(* LS Electric XG5000 project: 제일교회_조명제어 *)
(* PLC LSPLC *)
(* module base 0 slot 0: Cnet:XGL-C42A/B (Cnet 통신 모듈(RS-422/485, RS-422/485)) *)
(* module base 0 slot 1: 입력 모듈:XGI-D24A/B (DC 24V 입력, 32점 (전류소스 싱크공용/ 전류소스 입력)) *)
(* module base 0 slot 2: 입력 모듈:XGI-D21A (DC 24V 입력, 8점 (전류소스/싱크입력)) *)
(* module base 0 slot 3: 출력 모듈:XGQ-TR4A/B (트랜지스터 출력, 32점 (0.1A용, 싱크출력/소스출력)) *)

(* Comments on direct variables
%MX92	SET - 01_Button
%MX93	SET - 02_Button
%MX94	SET - 03_Button
%MX95	SET - 01_Lamp
%MX96	SET - 02_Lamp
%MX97	SET - 03_Lamp
%MX98	Reset
[SCADA]
%MX99	SHUT OFF
%MX100	MAIN POWER PBL
%MX101	십자가 PBL
%MX102	강대상 위 천정 PBL
%MX103	강대석(좌) PBL
%MX104	무대조명(좌) PBL
%MX105	(미정) PBL
%MX106	본당벽체 간접 PBL
%MX107	복도(좌) PBL
%MX108	중벽체(반달 좌) PBL
%MX109	중벽체 간접(좌) PBL
%MX110	기둥간접(좌) PBL
%MX111	중앙천정 강대상 PBL
%MX112	중앙천정앞(50W전구색) PBL
%MX113	중앙천정좌 간접 PBL
%MX114	중앙천정우 간접 PBL
%MX115	중앙천정U(20W주광색) PBL
%MX116	중앙천정뒤(50W전구색) PBL
%MX117	강대석 (우) PBL
%MX118	무대조명(우) PBL
%MX119	(미정) PBL
%MX120	본당벽체 간접 PBL
%MX121	복도(우) PBL
%MX122	중벽채(반달 우) PBL
%MX123	중벽체 간접(우) PBL
%MX124	기둥간접(우) PBL
%MX125	2층 후미 PBL
%MX126	종탑 PBL
%MX127	LAMP TEST PBL
%MX128	BUZZER STOP PBL[SR]
%MX129	RESET PBL[SR]
%MX130	SPARE
%MX131	SPARE
%MX160	Main Switch On
%MX161	성가대 P-S/W
%MX170	SCADA POWER PB [SCA]
%MX171	REMOTE POWER PB [SCA]
%MX192	십자가_SET [SCADA]
%MX193	강대상 위 천장_SET [SCADA]
%MX194	강대석 좌_SET [SCADA]
%MX195	무대조명(좌)_SET [SCADA]
%MX197	본당벽체-간접(좌)_SET [SCADA]
%MX198	복도(좌)_SET [SCADA]
%MX199	중벽체-반달(좌)_SET [SCADA]
%MX200	중벽체-간접(좌)_SET [SCADA]
%MX202	중앙천장 강대상_SET [SCADA]
%MX203	중앙천장앞_SET [SCADA]
%MX204	중앙천정좌 간접_SET [SCADA]
%MX205	중앙천장우 간접_SET [SCADA]
%MX206	중앙천정 U_SET [SCADA]
%MX207	중앙천정-뒤_SET [SCADA]
%MX208	강대석-우_SET [SCADA]
%MX209	무대조명(우)_SET [SCADA]
%MX211	본당벽체-간접(우)_SET [SCADA]
%MX212	복도(우)_SET [SCADA]
%MX213	중벽체-반달(우)_SET [SCADA]
%MX214	중벽체-간접 (우)_SET [SCADA]
%MX216	후미 중앙 기둥 간접등_SET [SCADA]
%MX217	종탑_SET [SCADA]
%MX284	BUZZER STOP [SCA]
%MX400	REMOTE POWER LAMP[REM]
%MX401	십자가 [REM]
%MX402	강대상 위 천정 [REM]
%MX403	강대석(좌) [REM]
%MX404	무대조명(좌) [REM]
%MX405	(미정) [REM]
%MX406	본당벽체 간접 [REM]
%MX407	복도 [REM]
%MX408	중벽체-반달(좌) [REM]
%MX409	중벽체 간접 [REM]
%MX410	기둥간접 [REM]
%MX411	중앙천정 강대상
[REM]
%MX412	중앙천정앞
50W전구색
[REM]
%MX413	중앙천정좌 간접 [REM]
%MX414	중앙천정우 간접 [REM]
%MX415	중앙천정U(20W주광색) [REM]
%MX416	중앙천정뒤(50W전구색) [REM]
%MX417	강대석 (우) [REM]
%MX418	무대조명(우) [REM]
%MX419	(미정) [REM]
%MX420	본당벽체 간접 [REM]
%MX421	복도 [REM]
%MX422	중벽채-반달(우) [REM]
%MX423	중벽체 간접 [REM]
%MX424	기둥간접 [REM]
%MX425	2층 후미 [REM]
%MX426	종탑 [REM]
%MX427	LAMP TEST [REM]
%MX428	BUZZER STOP [REM]
%MX429	RESET [REM]
%MX430	SPARE [REM]
%MX431	SPARE [REM]
%MX500	MAIN POWER LAMP
%MX501	십자가 LAMP
%MX502	강대상 위 천정 LAMP
%MX503	강대석(좌) LAMP
%MX504	무대조명(좌) LAMP
%MX505	(미정) LAMP
%MX506	본당벽체 간접 LAMP
%MX507	복도 LAMP
%MX508	중벽체(반달) LAMP
%MX509	중벽체 간접 LAMP
%MX510	기둥간접 LAMP
%MX511	중앙천정 강대상 LAMP
%MX512	중앙천정앞(50W전구색) LAMP
%MX513	중앙천정좌 간접 LAMP
%MX514	중앙천정우 간접 LAMP
%MX515	중앙천정U(20W주광색) LAMP
%MX516	중앙천정뒤(50W전구색) LAMP
%MX517	강대석 (우) LAMP
%MX518	무대조명(우) LAMP
%MX519	(미정) LAMP
%MX520	본당벽체 간접 LAMP
%MX521	복도 LAMP
%MX522	중벽채(반달) LAMP
%MX523	중벽체 간접 LAMP
%MX524	기둥간접 LAMP
%MX525	2층 후미 LAMP
%MX526	종탑 LAMP
%MX527	LAMP TEST LAMP
%MX528	BUZZER STOP LAMP
%MX529	RESET LAMP
%MX530	BUZZER
[[REM]]
%MX531	SPARE LAMP
%MX600	SCADA POWER LAMP_[SCA]
%MX601	십자가_S/W [SCADA]
%MX602	강대상 위 천장_S/W [SCADA]
%MX603	강대석 좌_S/W [SCADA]
%MX604	무대조명(좌)_S/W [SCADA]
%MX606	본당벽체-간접(좌)_S/W [SCADA]
%MX607	복도(좌)_S/W [SCADA]
%MX608	중벽체-반달(좌)_S/W [SCADA]
%MX609	중벽체-간접(좌)_S/W [SCADA]
%MX611	중앙천장 강대상_S/W [SCADA]
%MX612	중앙천장앞_S/W [SCADA]
%MX613	중앙천정좌 간접_S/W [SCADA]
%MX614	중앙천장우 간접_S/W [SCADA]
%MX615	중앙천정 U_S/W [SCADA]
%MX616	중앙천정-뒤_S/W [SCADA]
%MX617	강대석-우_S/W [SCADA]
%MX618	무대조명(우)_S/W [SCADA]
%MX620	본당벽체-간접(우)_S/W [SCADA]
%MX621	복도(우)_S/W [SCADA]
%MX622	중벽체-반달(우)_S/W [SCADA]
%MX623	중벽체-간접 (우)_S/W [SCADA]
%MX625	후미 중앙 기둥 간접등_S/W [SCADA]
%MX626	종탑_S/W [SCADA]
%MX640	중앙1열 OUT
%MX641	중앙2열 OUT
%MX642	중앙3열 OUT
%MX643	중앙4열 OUT
%MX644	중앙5열 OUT
%MX645	중앙6열 OUT
%MX646	중앙7열 OUT
%MX647	중앙8열 OUT
%MX648	중앙9열 OUT
%MX649	중앙10열 OUT
%MX650	장로석 OUT
%MX651	장로석 SPOT-OUT
%MX652	성가대 OUT
%MX653	성가대 SPOT-OUT
%MX654	좌측통로 OUT
%MX655	우측통로 OUT
%MX656	후단1열 OUT
%MX657	후단2열 OUT
%MX658	후단3열 OUT
%MX659	종탑 OUT
%MX704	십자가_[SET]_OUT [SCADA]
%MX705	강대상 위 천장_[SET]_OUT [SCADA]
%MX706	강대석 좌_[SET]_OUT [SCADA]
%MX707	무대조명(좌)_[SET]_OUT [SCADA]
%MX709	본당벽체-간접(좌)_[SET]_OUT [SCADA]
%MX710	복도(좌)_[SET]_OUT [SCADA]
%MX711	중벽체-반달(좌)_[SET]_OUT [SCADA]
%MX712	중벽체-간접(좌)_[SET]_OUT [SCADA]
%MX714	중앙천장 강대상_[SET]_OUT [SCADA]
%MX715	중앙천장앞_[SET]_OUT [SCADA]
%MX716	중앙천정좌 간접_[SET]_OUT [SCADA]
%MX717	중앙천장우 간접_[SET]_OUT [SCADA]
%MX718	중앙천정 U_[SET]_OUT [SCADA]
%MX719	중앙천정-뒤_[SET]_OUT [SCADA]
%MX720	강대석-우_[SET]_OUT [SCADA]
%MX721	무대조명(우)_[SET]_OUT [SCADA]
%MX723	본당벽체-간접(우)_[SET]_OUT [SCADA]
%MX724	복도(우)_[SET]_OUT [SCADA]
%MX725	중벽체-반달(우)_[SET]_OUT [SCADA]
%MX726	중벽체-간접 (우)_[SET]_OUT [SCADA]
%MX728	후미 중앙 기둥 간접등_[SET]_OUT [SCADA]
%MX729	종탑_[SET]_OUT [SCADA]
%MX800	십자가_S/W_OUT [SCADA]
%MX801	강대상 위 천장_S/W_OUT [SCADA]
%MX802	강대석 좌_S/W_OUT [SCADA]
%MX803	무대조명(좌)_S/W_OUT [SCADA]
%MX805	본당벽체-간접(좌)_S/W_OUT [SCADA]
%MX806	복도(좌)_S/W_OUT [SCADA]
%MX807	중벽체-반달(좌)_S/W_OUT [SCADA]
%MX808	중벽체-간접(좌)_S/W_OUT [SCADA]
%MX810	중앙천장 강대상_S/W_OUT [SCADA]
%MX811	중앙천장앞_S/W_OUT [SCADA]
%MX812	중앙천정좌 간접_S/W_OUT [SCADA]
%MX813	중앙천장우 간접_S/W_OUT [SCADA]
%MX814	중앙천정 U_S/W_OUT [SCADA]
%MX815	중앙천정-뒤_S/W_OUT [SCADA]
%MX816	강대석-우_S/W_OUT [SCADA]
%MX817	무대조명(우)_S/W_OUT [SCADA]
%MX819	본당벽체-간접(우)_S/W_OUT [SCADA]
%MX820	복도(우)_S/W_OUT [SCADA]
%MX821	중벽체-반달(우)_S/W_OUT [SCADA]
%MX822	중벽체-간접 (우)_S/W_OUT [SCADA]
%MX824	후미 중앙 기둥 간접등_S/W_OUT [SCADA]
%MX825	종탑_S/W_OUT [SCADA]
%MX911	Total Alarm
%MX992	중앙1열 S/W
%MX993	중앙2열 S/W
%MX994	중앙3열 S/W
%MX995	중앙4열 S/W
%MX996	중앙5열 S/W
%MX997	중앙6열 S/W
%MX998	중앙7열 S/W
%MX999	중앙8열 S/W
%MX1000	중앙9열 S/W
%MX1001	중앙10열 S/W
%MX1002	장로석 S/W
%MX1003	장로석 SPOT S/W
%MX1004	성가대 S/W
%MX1005	성가대 SPOT S/W [MAIN]
%MX1006	좌측통로 S/W
%MX1007	우측통로 S/W
%MX1008	후단1열 S/W
%MX1009	후단2열 S/W
%MX1010	후단3열 S/W
%MX1011	종탑 S/W
%MX1040	중앙1열 M/C-a
%MX1041	중앙2열 M/C-a
%MX1042	중앙3열 M/C-a
%MX1043	중앙4열 M/C-a
%MX1044	중앙5열 M/C-a
%MX1045	중앙6열 M/C-a
%MX1046	중앙7열 M/C-a
%MX1047	중앙8열 M/C-a
%MX1048	중앙9열 M/C-a
%MX1049	중앙10열 M/C-a
%MX1050	장로석 M/C-a
%MX1051	장로석 SPOT M/C-a
%MX1052	성가대 M/C-a
%MX1053	성가대 SPOT M/C-a
%MX1054	좌측통로 M/C-a
%MX1055	우측통로 M/C-a
%MX1056	후단1열 M/C-a
%MX1057	후단2열 M/C-a
%MX1058	후단3열 M/C-a
%MX1059	종탑 M/C-a
%MW0	IN-COM0
%MW1	IN-COM1
%MW2	OUT-COM0
%MW3	OUT-COM1
%MW4	Reset-Word
%MW12	Reset-Word
%MD22	SET_OUT
%MD31	MAIN_SW
%QX0.3.0	중앙1열
%QX0.3.1	중앙2열
%QX0.3.2	중앙3열
%QX0.3.3	중앙4열
%QX0.3.4	중앙5열
%QX0.3.5	중앙6열
%QX0.3.6	중앙7열
%QX0.3.7	중앙8열
%QX0.3.8	중앙9열
%QX0.3.9	중앙10열
%QX0.3.10	장로석
%QX0.3.11	장로석 SPOT
%QX0.3.12	성가대
%QX0.3.13	성가대 SPOT
%QX0.3.14	좌측통로
%QX0.3.15	우측통로
%QX0.3.16	후단1열
%QX0.3.17	후단2열
%QX0.3.18	후단3열
%QX0.3.19	종탑
%QX0.3.20	BUZZER
[MAIN]
%IX0.1.0	중앙1열 S/W
%IX0.1.1	중앙2열 S/W
%IX0.1.2	중앙3열 S/W
%IX0.1.3	중앙4열 S/W
%IX0.1.4	중앙5열 S/W
%IX0.1.5	중앙6열 S/W
%IX0.1.6	중앙7열 S/W
%IX0.1.7	중앙8열 S/W
%IX0.1.8	중앙9열 S/W
%IX0.1.9	중앙10열 S/W
%IX0.1.10	장로석 S/W
%IX0.1.11	장로석 SPOT S/W
%IX0.1.12	성가대 S/W
%IX0.1.13	성가대 SPOT S/W
%IX0.1.14	좌측통로 S/W
%IX0.1.15	우측통로 S/W
%IX0.1.16	후단1열 S/W
%IX0.1.17	후단2열 S/W
%IX0.1.18	후단3열 S/W
%IX0.1.19	종탑
%IX0.1.20	중앙1열 M/C-a
%IX0.1.21	중앙2열 M/C-a
%IX0.1.22	중앙3열 M/C-a
%IX0.1.23	중앙4열 M/C-a
%IX0.1.24	중앙5열 M/C-a
%IX0.1.25	중앙6열 M/C-a
%IX0.1.26	중앙7열 M/C-a
%IX0.1.27	중앙8열 M/C-a
%IX0.1.28	중앙9열 M/C-a
%IX0.1.29	중앙10열 M/C-a
%IX0.1.30	장로석 M/C-a
%IX0.1.31	장로석 SPOT M/C-a
%IX0.2.0	성가대 M/C-a
%IX0.2.1	성가대 SPOT M/C-a
%IX0.2.2	좌측통로 M/C-a
%IX0.2.3	우측통로 M/C-a
%IX0.2.4	후단1열 M/C-a
%IX0.2.5	후단2열 M/C-a
%IX0.2.6	후단3열 M/C-a
%IX0.2.7	종탑
M/C-a
*)

FUNCTION_BLOCK SET_FF
VAR_INPUT
    IN : BOOL;
    RESET : BOOL;
    CHECK_SET : BOOL;
END_VAR
VAR_IN_OUT
    SET : BOOL;
    MANUAL : BOOL;
END_VAR
VAR_OUTPUT
    FF : BOOL;
END_VAR
VAR
    IN_COIL : BOOL;
END_VAR
VAR
    _e1 : R_TRIG;
    _e2 : R_TRIG;
END_VAR

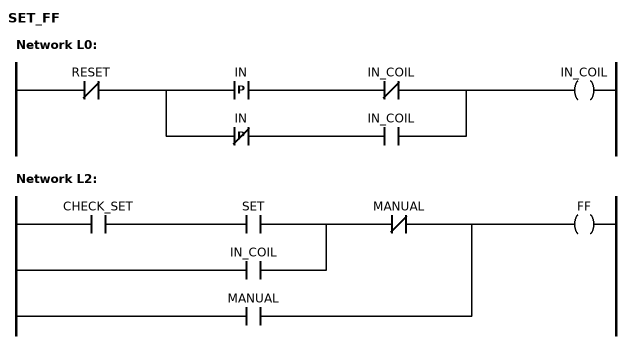
(* Rung L0 *)
_e1(CLK := IN);
_e2(CLK := IN);
IN_COIL := NOT RESET AND ((_e1.Q AND NOT IN_COIL) OR (NOT _e2.Q AND IN_COIL));
(* Rung L2 *)
FF := (((CHECK_SET AND SET) OR IN_COIL) AND NOT MANUAL) OR MANUAL;
END_FUNCTION_BLOCK

PROGRAM Remote (* task: 스캔 프로그램 *)
VAR
    INST : FF;
    INST1 : FF;
    IN_0_HIGH : BYTE;
    IN_0_LOW : BYTE;
    IN_1_HIGH : BYTE;
    IN_1_LOW : BYTE;
    OUT_0_HIGH : BYTE;
    OUT_0_LOW : BYTE;
    remote_holding : BOOL;
END_VAR

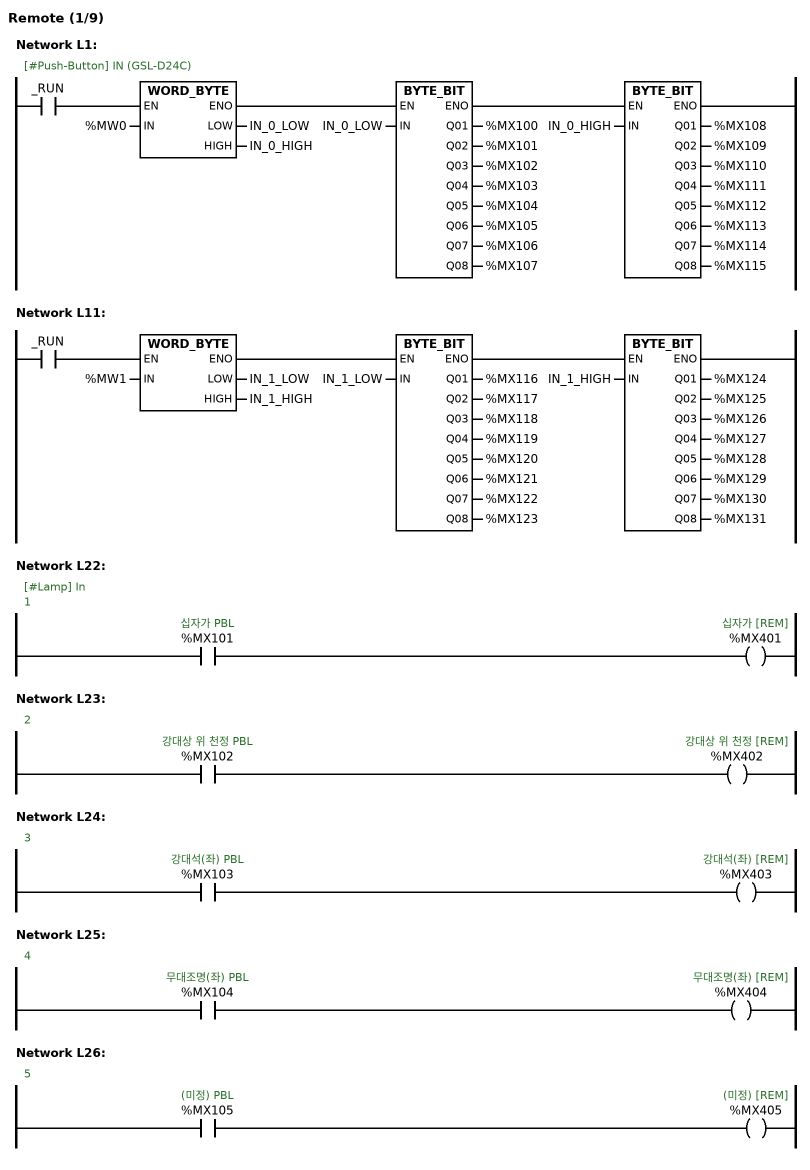
(* [#Push-Button] IN (GSL-D24C) *)
(* Rung L1 *)
IF _RUN THEN
    IN_0_LOW := WORD_BYTE(IN := %MW0, HIGH => IN_0_HIGH);
    %MX100 := BYTE_BIT(IN := IN_0_LOW, Q02 => %MX101, Q03 => %MX102, Q04 => %MX103, Q05 => %MX104, Q06 => %MX105, Q07 => %MX106, Q08 => %MX107);
    %MX108 := BYTE_BIT(IN := IN_0_HIGH, Q02 => %MX109, Q03 => %MX110, Q04 => %MX111, Q05 => %MX112, Q06 => %MX113, Q07 => %MX114, Q08 => %MX115);
END_IF;
(* Rung L11 *)
IF _RUN THEN
    IN_1_LOW := WORD_BYTE(IN := %MW1, HIGH => IN_1_HIGH);
    %MX116 := BYTE_BIT(IN := IN_1_LOW, Q02 => %MX117, Q03 => %MX118, Q04 => %MX119, Q05 => %MX120, Q06 => %MX121, Q07 => %MX122, Q08 => %MX123);
    %MX124 := BYTE_BIT(IN := IN_1_HIGH, Q02 => %MX125, Q03 => %MX126, Q04 => %MX127, Q05 => %MX128, Q06 => %MX129, Q07 => %MX130, Q08 => %MX131);
END_IF;
(* [#Lamp] In *)
(* Rung L22 *)
%MX401 := %MX101;
(* 1 *)
(* Rung L23 *)
%MX402 := %MX102;
(* 2 *)
(* Rung L24 *)
%MX403 := %MX103;
(* 3 *)
(* Rung L25 *)
%MX404 := %MX104;
(* 4 *)
(* Rung L26 *)
%MX405 := %MX105;
(* 5 *)

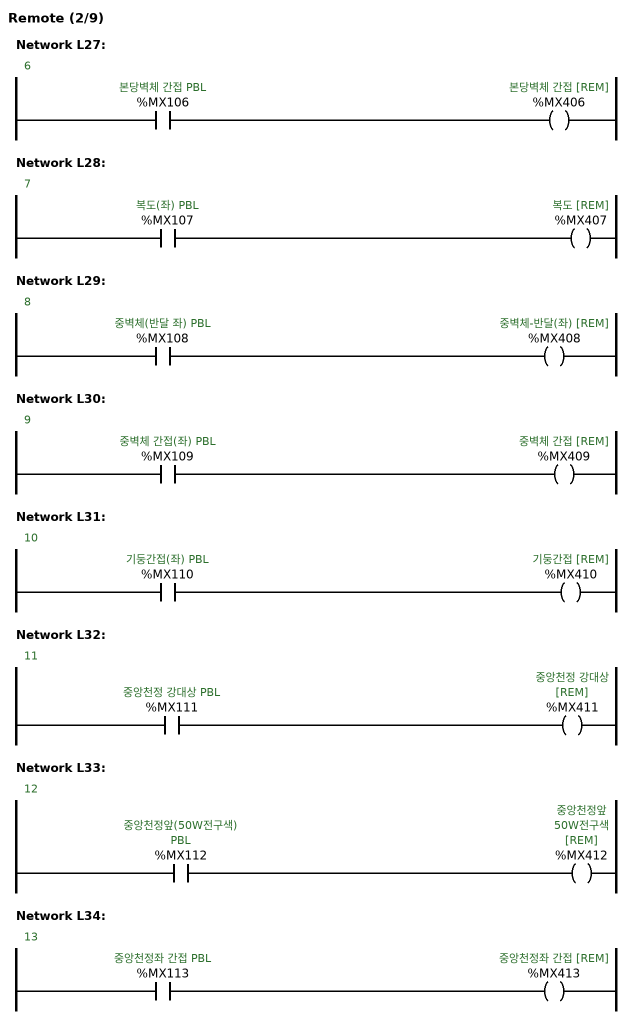
(* Rung L27 *)
%MX406 := %MX106;
(* 6 *)
(* Rung L28 *)
%MX407 := %MX107;
(* 7 *)
(* Rung L29 *)
%MX408 := %MX108;
(* 8 *)
(* Rung L30 *)
%MX409 := %MX109;
(* 9 *)
(* Rung L31 *)
%MX410 := %MX110;
(* 10 *)
(* Rung L32 *)
%MX411 := %MX111;
(* 11 *)
(* Rung L33 *)
%MX412 := %MX112;
(* 12 *)
(* Rung L34 *)
%MX413 := %MX113;
(* 13 *)

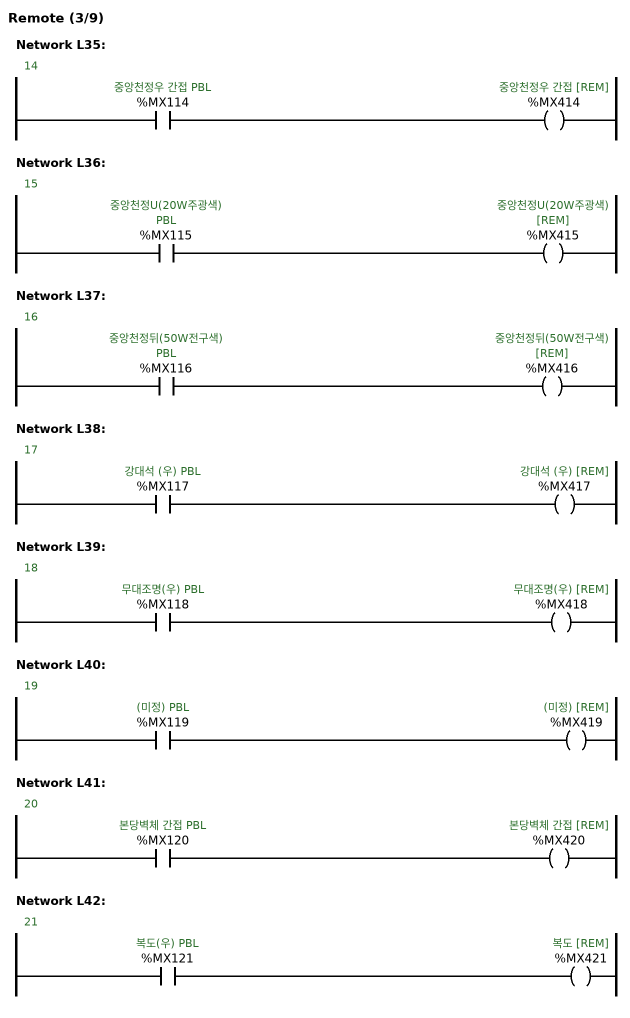
(* Rung L35 *)
%MX414 := %MX114;
(* 14 *)
(* Rung L36 *)
%MX415 := %MX115;
(* 15 *)
(* Rung L37 *)
%MX416 := %MX116;
(* 16 *)
(* Rung L38 *)
%MX417 := %MX117;
(* 17 *)
(* Rung L39 *)
%MX418 := %MX118;
(* 18 *)
(* Rung L40 *)
%MX419 := %MX119;
(* 19 *)
(* Rung L41 *)
%MX420 := %MX120;
(* 20 *)
(* Rung L42 *)
%MX421 := %MX121;
(* 21 *)

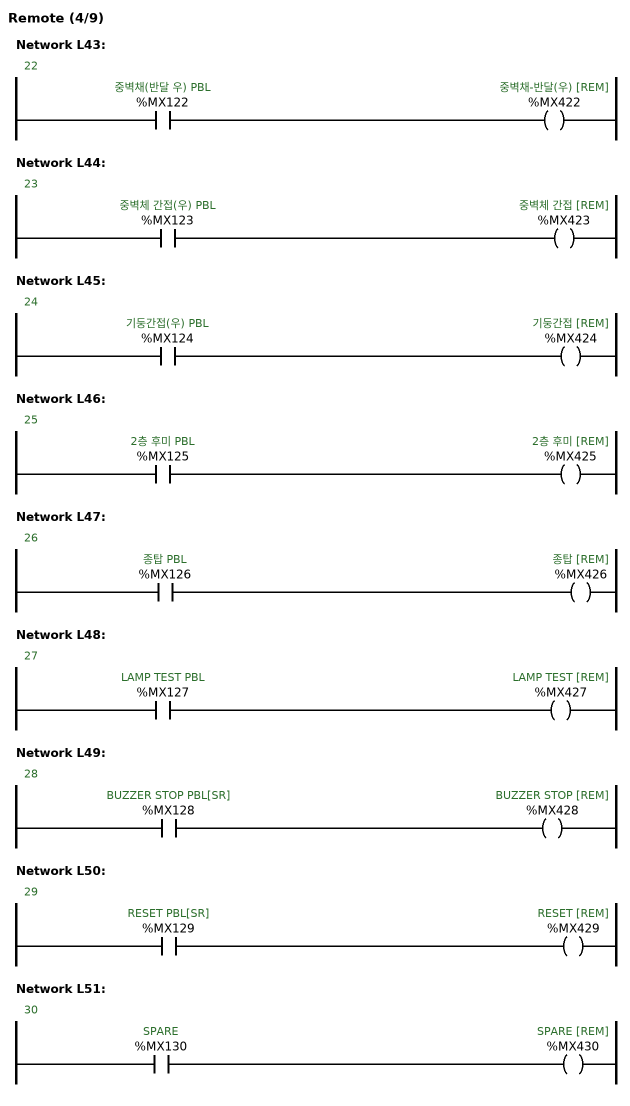
(* Rung L43 *)
%MX422 := %MX122;
(* 22 *)
(* Rung L44 *)
%MX423 := %MX123;
(* 23 *)
(* Rung L45 *)
%MX424 := %MX124;
(* 24 *)
(* Rung L46 *)
%MX425 := %MX125;
(* 25 *)
(* Rung L47 *)
%MX426 := %MX126;
(* 26 *)
(* Rung L48 *)
%MX427 := %MX127;
(* 27 *)
(* Rung L49 *)
%MX428 := %MX128;
(* 28 *)
(* Rung L50 *)
%MX429 := %MX129;
(* 29 *)
(* Rung L51 *)
%MX430 := %MX130;
(* 30 *)

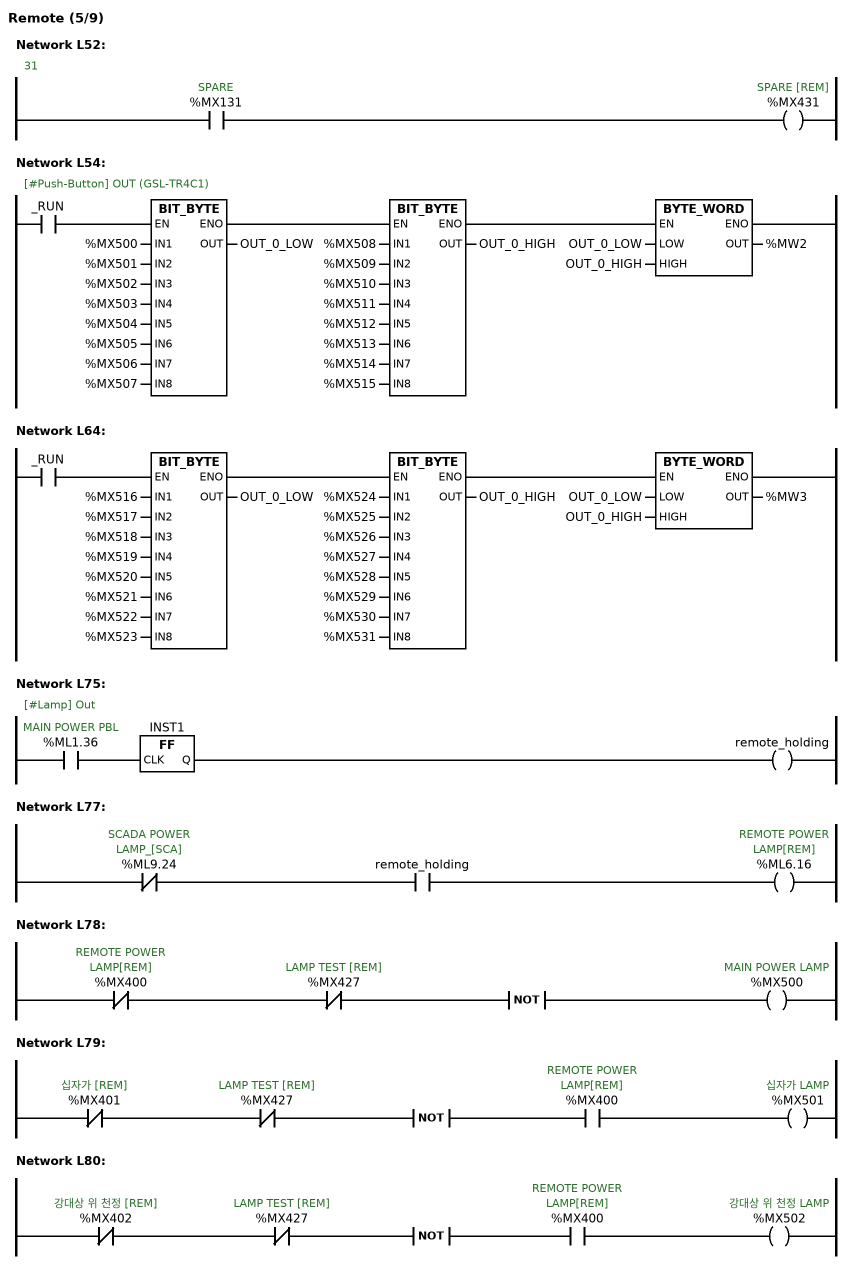
(* Rung L52 *)
%MX431 := %MX131;
(* 31 *)
(* [#Push-Button] OUT (GSL-TR4C1) *)
(* Rung L54 *)
IF _RUN THEN
    OUT_0_LOW := BIT_BYTE(%MX500, %MX501, %MX502, %MX503, %MX504, %MX505, %MX506, %MX507);
    OUT_0_HIGH := BIT_BYTE(%MX508, %MX509, %MX510, %MX511, %MX512, %MX513, %MX514, %MX515);
    %MW2 := BYTE_WORD(LOW := OUT_0_LOW, HIGH := OUT_0_HIGH);
END_IF;
(* Rung L64 *)
IF _RUN THEN
    OUT_0_LOW := BIT_BYTE(%MX516, %MX517, %MX518, %MX519, %MX520, %MX521, %MX522, %MX523);
    OUT_0_HIGH := BIT_BYTE(%MX524, %MX525, %MX526, %MX527, %MX528, %MX529, %MX530, %MX531);
    %MW3 := BYTE_WORD(LOW := OUT_0_LOW, HIGH := OUT_0_HIGH);
END_IF;
(* [#Lamp] Out *)
(* Rung L75 *)
INST1(CLK := %ML1.36);
remote_holding := INST1.Q;
(* Rung L77 *)
%ML6.16 := NOT %ML9.24 AND remote_holding;
(* Rung L78 *)
%MX500 := NOT (NOT %MX400 AND NOT %MX427);
(* Rung L79 *)
%MX501 := NOT (NOT %MX401 AND NOT %MX427) AND %MX400;
(* Rung L80 *)
%MX502 := NOT (NOT %MX402 AND NOT %MX427) AND %MX400;

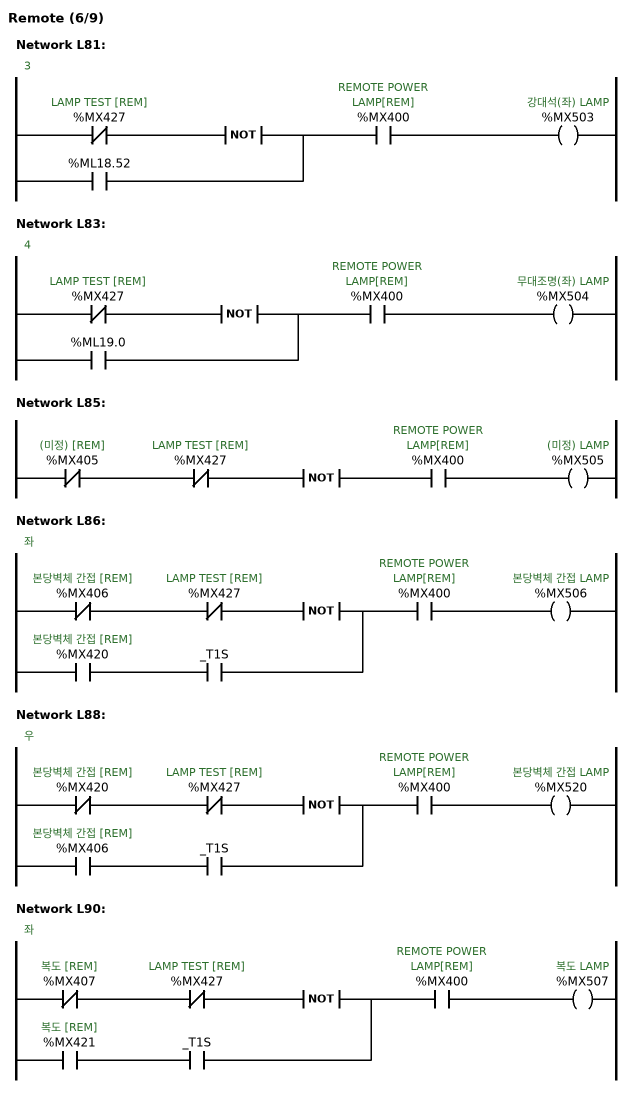
(* Rung L81 *)
%MX503 := (%MX427 OR %ML18.52) AND %MX400;
(* 3 *)
(* Rung L83 *)
%MX504 := (%MX427 OR %ML19.0) AND %MX400;
(* 4 *)
(* Rung L85 *)
%MX505 := NOT (NOT %MX405 AND NOT %MX427) AND %MX400;
(* Rung L86 *)
%MX506 := (NOT (NOT %MX406 AND NOT %MX427) OR (%MX420 AND _T1S)) AND %MX400;
(* 좌 *)
(* Rung L88 *)
%MX520 := (NOT (NOT %MX420 AND NOT %MX427) OR (%MX406 AND _T1S)) AND %MX400;
(* 우 *)
(* Rung L90 *)
%MX507 := (NOT (NOT %MX407 AND NOT %MX427) OR (%MX421 AND _T1S)) AND %MX400;
(* 좌 *)

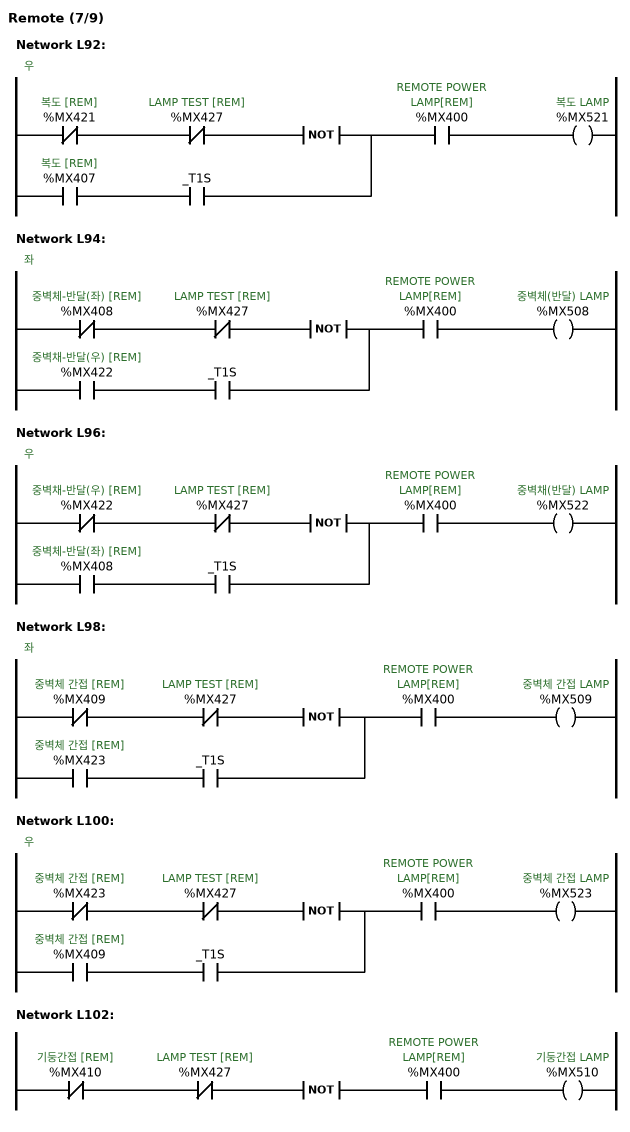
(* Rung L92 *)
%MX521 := (NOT (NOT %MX421 AND NOT %MX427) OR (%MX407 AND _T1S)) AND %MX400;
(* 우 *)
(* Rung L94 *)
%MX508 := (NOT (NOT %MX408 AND NOT %MX427) OR (%MX422 AND _T1S)) AND %MX400;
(* 좌 *)
(* Rung L96 *)
%MX522 := (NOT (NOT %MX422 AND NOT %MX427) OR (%MX408 AND _T1S)) AND %MX400;
(* 우 *)
(* Rung L98 *)
%MX509 := (NOT (NOT %MX409 AND NOT %MX427) OR (%MX423 AND _T1S)) AND %MX400;
(* 좌 *)
(* Rung L100 *)
%MX523 := (NOT (NOT %MX423 AND NOT %MX427) OR (%MX409 AND _T1S)) AND %MX400;
(* 우 *)
(* Rung L102 *)
%MX510 := NOT (NOT %MX410 AND NOT %MX427) AND %MX400;

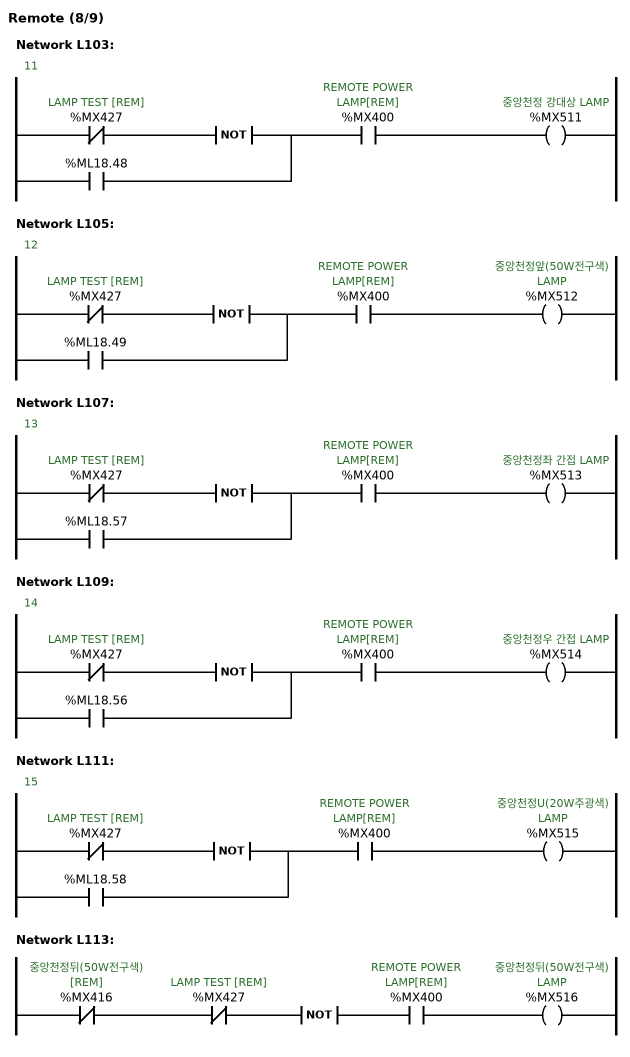
(* Rung L103 *)
%MX511 := (%MX427 OR %ML18.48) AND %MX400;
(* 11 *)
(* Rung L105 *)
%MX512 := (%MX427 OR %ML18.49) AND %MX400;
(* 12 *)
(* Rung L107 *)
%MX513 := (%MX427 OR %ML18.57) AND %MX400;
(* 13 *)
(* Rung L109 *)
%MX514 := (%MX427 OR %ML18.56) AND %MX400;
(* 14 *)
(* Rung L111 *)
%MX515 := (%MX427 OR %ML18.58) AND %MX400;
(* 15 *)
(* Rung L113 *)
%MX516 := NOT (NOT %MX416 AND NOT %MX427) AND %MX400;

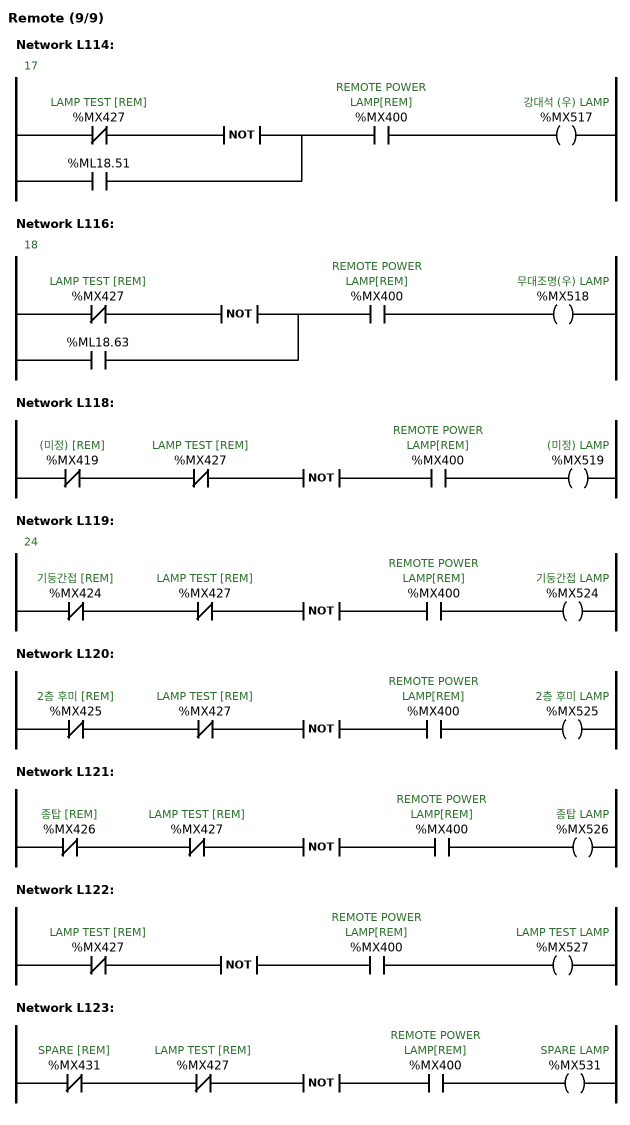
(* Rung L114 *)
%MX517 := (%MX427 OR %ML18.51) AND %MX400;
(* 17 *)
(* Rung L116 *)
%MX518 := (%MX427 OR %ML18.63) AND %MX400;
(* 18 *)
(* Rung L118 *)
%MX519 := NOT (NOT %MX419 AND NOT %MX427) AND %MX400;
(* Rung L119 *)
%MX524 := NOT (NOT %MX424 AND NOT %MX427) AND %MX400;
(* 24 *)
(* Rung L120 *)
%MX525 := NOT (NOT %MX425 AND NOT %MX427) AND %MX400;
(* Rung L121 *)
%MX526 := NOT (NOT %MX426 AND NOT %MX427) AND %MX400;
(* Rung L122 *)
%MX527 := %MX427 AND %MX400;
(* Rung L123 *)
%MX531 := NOT (NOT %MX431 AND NOT %MX427) AND %MX400;
END_PROGRAM

PROGRAM SCADA (* task: 스캔 프로그램 *)
VAR
    INST : FF;
    INST1 : FF;
    INST2 : FF;
    INST3 : FF;
    IN_0_HIGH : BYTE;
    IN_0_LOW : BYTE;
    IN_1_HIGH : BYTE;
    IN_1_LOW : BYTE;
END_VAR
VAR
    _e1 : R_TRIG;
    _e2 : R_TRIG;
END_VAR

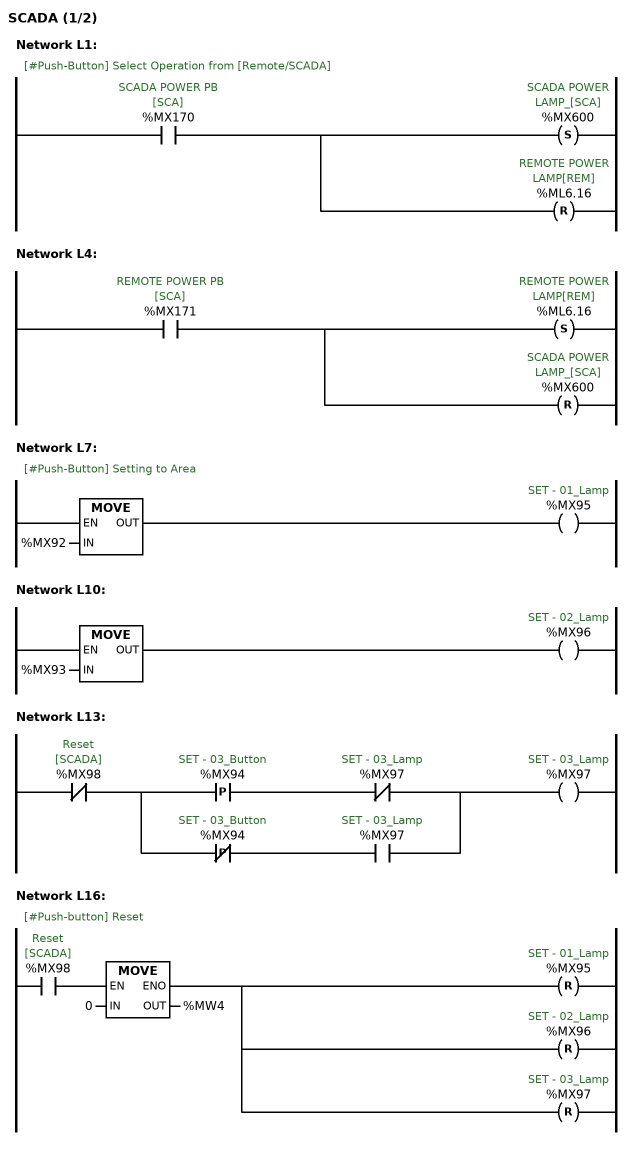
(* [#Push-Button] Select Operation from [Remote/SCADA] *)
(* Rung L1 *)
IF %MX170 THEN
    %MX600 := TRUE;
    %ML6.16 := FALSE;
END_IF;
(* Rung L4 *)
IF %MX171 THEN
    %ML6.16 := TRUE;
    %MX600 := FALSE;
END_IF;
(* [#Push-Button] Setting to Area *)
(* Rung L7 *)
%MX95 := %MX92;
(* Rung L10 *)
%MX96 := %MX93;
(* Rung L13 *)
_e1(CLK := %MX94);
_e2(CLK := %MX94);
%MX97 := NOT %MX98 AND ((_e1.Q AND NOT %MX97) OR (NOT _e2.Q AND %MX97));
(* [#Push-button] Reset *)
(* Rung L16 *)
IF %MX98 THEN
    %MW4 := 0;
    %MX95 := FALSE;
    %MX96 := FALSE;
    %MX97 := FALSE;
END_IF;

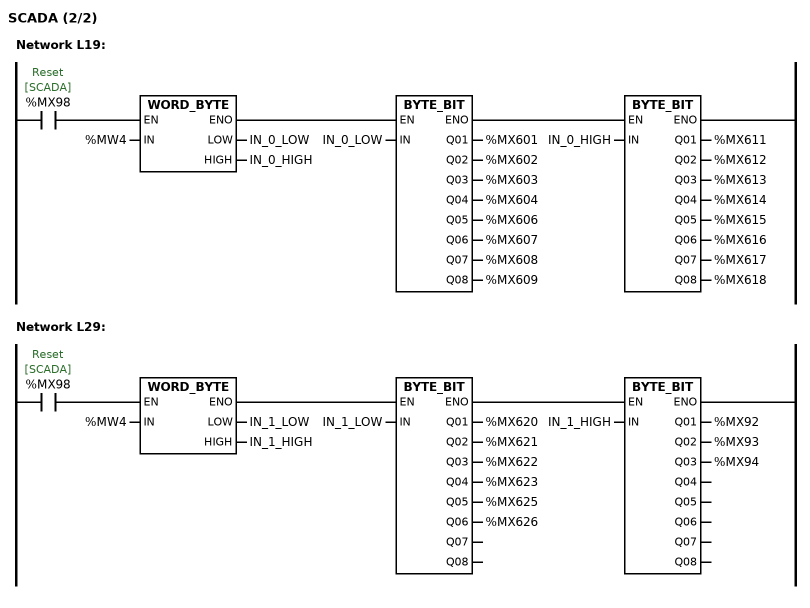
(* Rung L19 *)
IF %MX98 THEN
    IN_0_LOW := WORD_BYTE(IN := %MW4, HIGH => IN_0_HIGH);
    %MX601 := BYTE_BIT(IN := IN_0_LOW, Q02 => %MX602, Q03 => %MX603, Q04 => %MX604, Q05 => %MX606, Q06 => %MX607, Q07 => %MX608, Q08 => %MX609);
    %MX611 := BYTE_BIT(IN := IN_0_HIGH, Q02 => %MX612, Q03 => %MX613, Q04 => %MX614, Q05 => %MX615, Q06 => %MX616, Q07 => %MX617, Q08 => %MX618);
END_IF;
(* Rung L29 *)
IF %MX98 THEN
    IN_1_LOW := WORD_BYTE(IN := %MW4, HIGH => IN_1_HIGH);
    %MX620 := BYTE_BIT(IN := IN_1_LOW, Q02 => %MX621, Q03 => %MX622, Q04 => %MX623, Q05 => %MX625, Q06 => %MX626);
    %MX92 := BYTE_BIT(IN := IN_1_HIGH, Q02 => %MX93, Q03 => %MX94);
END_IF;
END_PROGRAM

PROGRAM Main_Program (* task: 스캔 프로그램 *)
VAR
    INST : FF;
    INST1 : FF;
    INST10 : FF;
    INST11 : FF;
    INST12 : FF;
    INST13 : FF;
    INST14 : FF;
    INST15 : FF;
    INST2 : FF;
    INST3 : FF;
    INST4 : FF;
    INST5 : FF;
    INST6 : FF;
    INST7 : FF;
    INST8 : FF;
    INST9 : FF;
END_VAR
VAR RETAIN
    INST16 : SET_FF;
    INST17 : SET_FF;
    INST18 : SET_FF;
    INST19 : SET_FF;
END_VAR

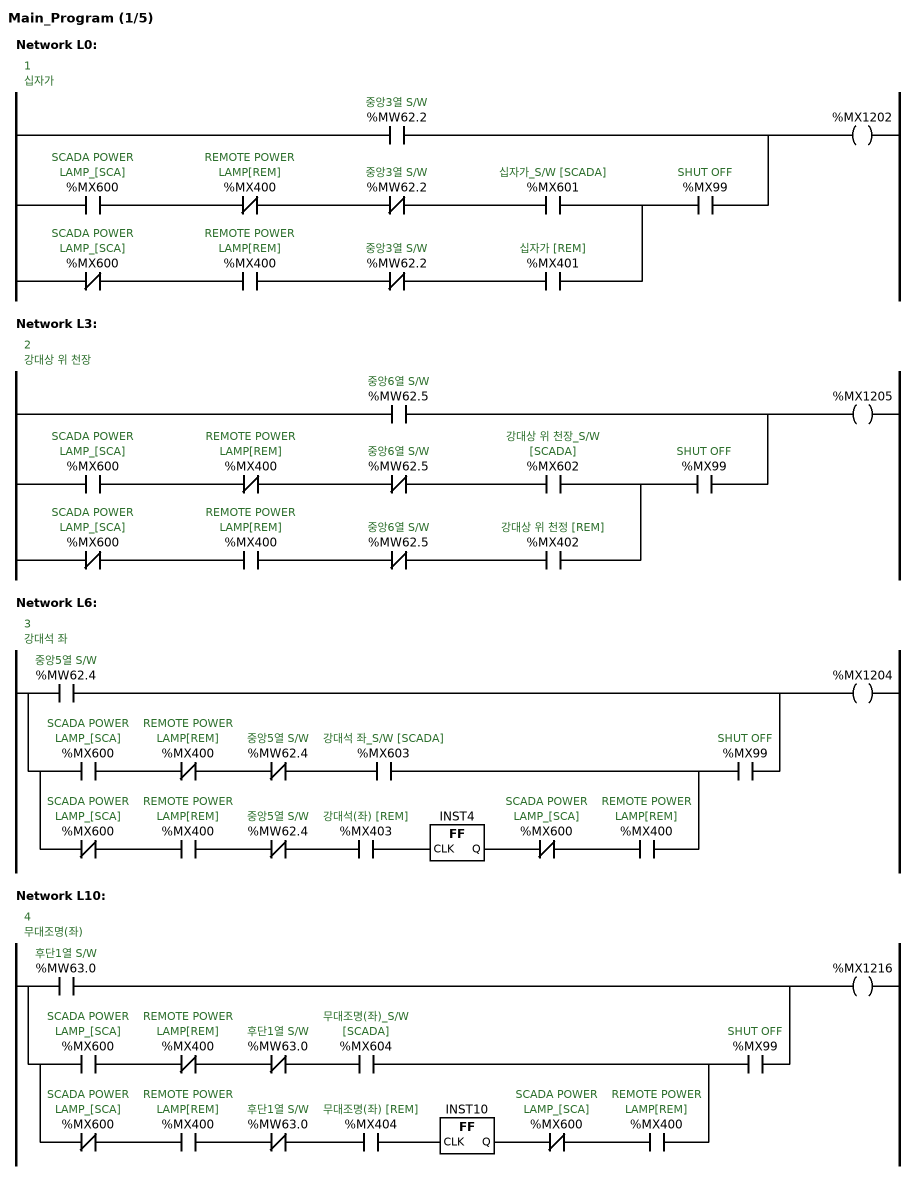
(* Rung L0 *)
%MX1202 := %MW62.2 OR (((%MX600 AND NOT %MX400 AND NOT %MW62.2 AND %MX601) OR (NOT %MX600 AND %MX400 AND NOT %MW62.2 AND %MX401)) AND %MX99);
(* 1 / 십자가 *)
(* Rung L3 *)
%MX1205 := %MW62.5 OR (((%MX600 AND NOT %MX400 AND NOT %MW62.5 AND %MX602) OR (NOT %MX600 AND %MX400 AND NOT %MW62.5 AND %MX402)) AND %MX99);
(* 2 / 강대상 위 천장 *)
(* Rung L6 *)
INST4(CLK := NOT %MX600 AND %MX400 AND NOT %MW62.4 AND %MX403);
%MX1204 := %MW62.4 OR (((%MX600 AND NOT %MX400 AND NOT %MW62.4 AND %MX603) OR (INST4.Q AND NOT %MX600 AND %MX400)) AND %MX99);
(* 3 / 강대석 좌 *)
(* Rung L10 *)
INST10(CLK := NOT %MX600 AND %MX400 AND NOT %MW63.0 AND %MX404);
%MX1216 := %MW63.0 OR (((%MX600 AND NOT %MX400 AND NOT %MW63.0 AND %MX604) OR (INST10.Q AND NOT %MX600 AND %MX400)) AND %MX99);
(* 4 / 무대조명(좌) *)

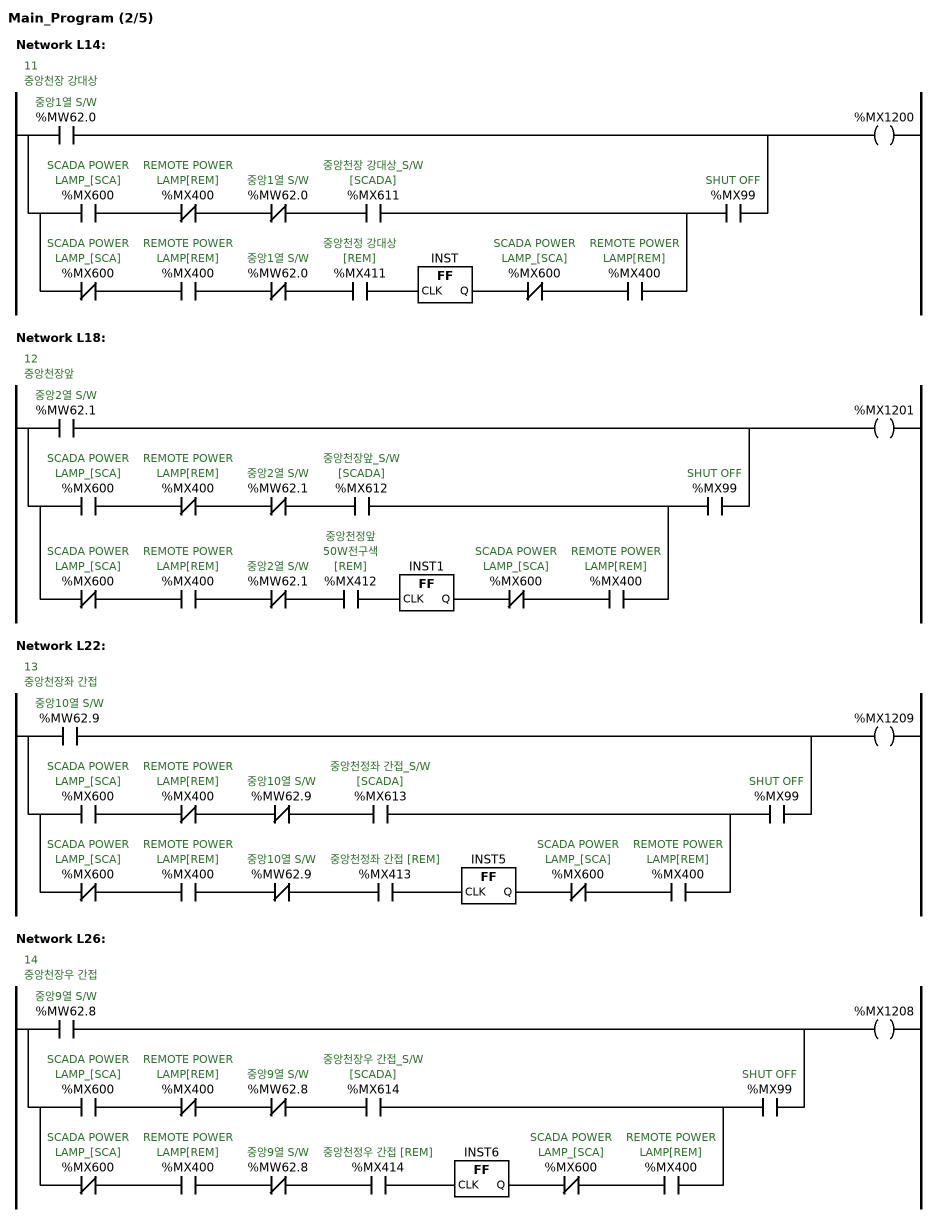
(* Rung L14 *)
INST(CLK := NOT %MX600 AND %MX400 AND NOT %MW62.0 AND %MX411);
%MX1200 := %MW62.0 OR (((%MX600 AND NOT %MX400 AND NOT %MW62.0 AND %MX611) OR (INST.Q AND NOT %MX600 AND %MX400)) AND %MX99);
(* 11 / 중앙천장 강대상 *)
(* Rung L18 *)
INST1(CLK := NOT %MX600 AND %MX400 AND NOT %MW62.1 AND %MX412);
%MX1201 := %MW62.1 OR (((%MX600 AND NOT %MX400 AND NOT %MW62.1 AND %MX612) OR (INST1.Q AND NOT %MX600 AND %MX400)) AND %MX99);
(* 12 / 중앙천장앞 *)
(* Rung L22 *)
INST5(CLK := NOT %MX600 AND %MX400 AND NOT %MW62.9 AND %MX413);
%MX1209 := %MW62.9 OR (((%MX600 AND NOT %MX400 AND NOT %MW62.9 AND %MX613) OR (INST5.Q AND NOT %MX600 AND %MX400)) AND %MX99);
(* 13 / 중앙천장좌 간접 *)
(* Rung L26 *)
INST6(CLK := NOT %MX600 AND %MX400 AND NOT %MW62.8 AND %MX414);
%MX1208 := %MW62.8 OR (((%MX600 AND NOT %MX400 AND NOT %MW62.8 AND %MX614) OR (INST6.Q AND NOT %MX600 AND %MX400)) AND %MX99);
(* 14 / 중앙천장우 간접 *)

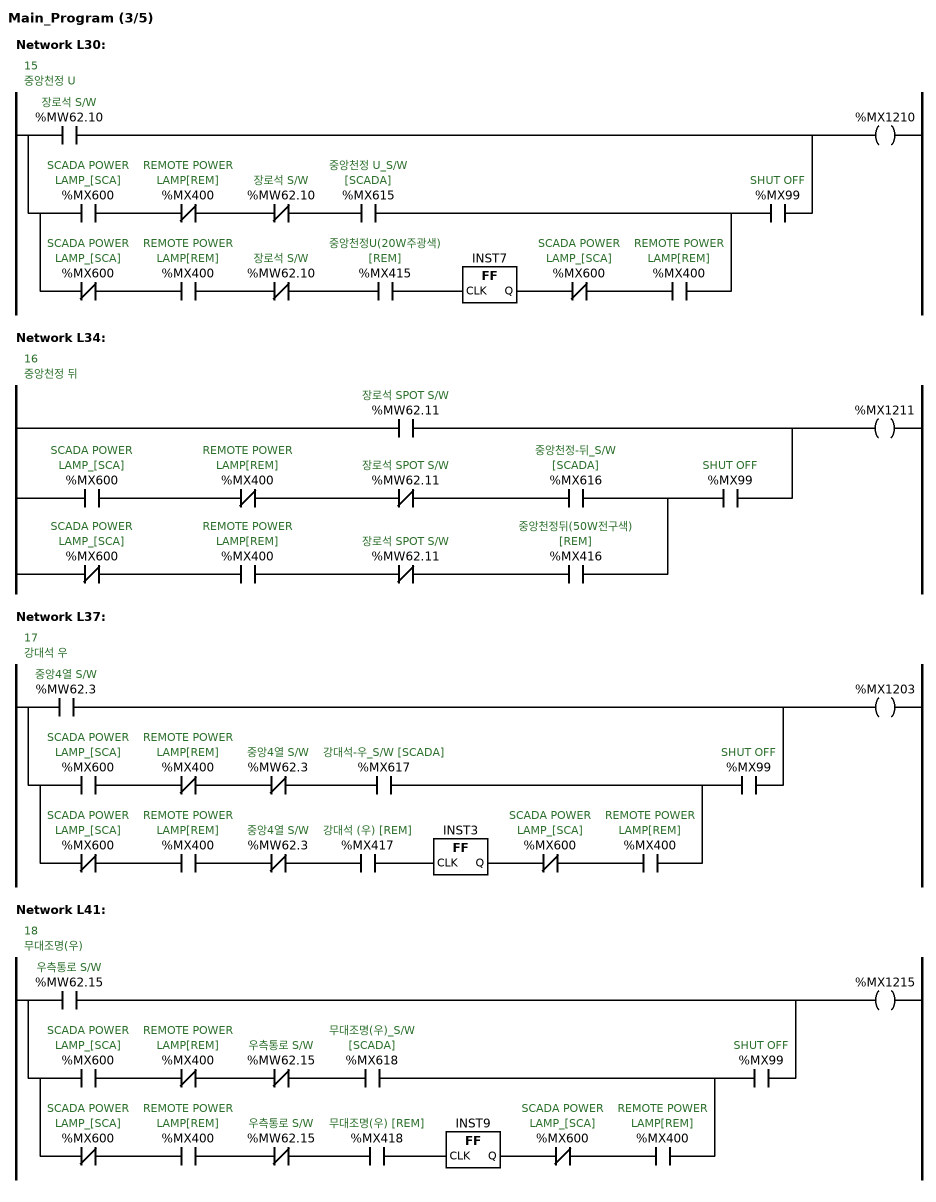
(* Rung L30 *)
INST7(CLK := NOT %MX600 AND %MX400 AND NOT %MW62.10 AND %MX415);
%MX1210 := %MW62.10 OR (((%MX600 AND NOT %MX400 AND NOT %MW62.10 AND %MX615) OR (INST7.Q AND NOT %MX600 AND %MX400)) AND %MX99);
(* 15 / 중앙천정 U *)
(* Rung L34 *)
%MX1211 := %MW62.11 OR (((%MX600 AND NOT %MX400 AND NOT %MW62.11 AND %MX616) OR (NOT %MX600 AND %MX400 AND NOT %MW62.11 AND %MX416)) AND %MX99);
(* 16 / 중앙천정 뒤 *)
(* Rung L37 *)
INST3(CLK := NOT %MX600 AND %MX400 AND NOT %MW62.3 AND %MX417);
%MX1203 := %MW62.3 OR (((%MX600 AND NOT %MX400 AND NOT %MW62.3 AND %MX617) OR (INST3.Q AND NOT %MX600 AND %MX400)) AND %MX99);
(* 17 / 강대석 우 *)
(* Rung L41 *)
INST9(CLK := NOT %MX600 AND %MX400 AND NOT %MW62.15 AND %MX418);
%MX1215 := %MW62.15 OR (((%MX600 AND NOT %MX400 AND NOT %MW62.15 AND %MX618) OR (INST9.Q AND NOT %MX600 AND %MX400)) AND %MX99);
(* 18 / 무대조명(우) *)

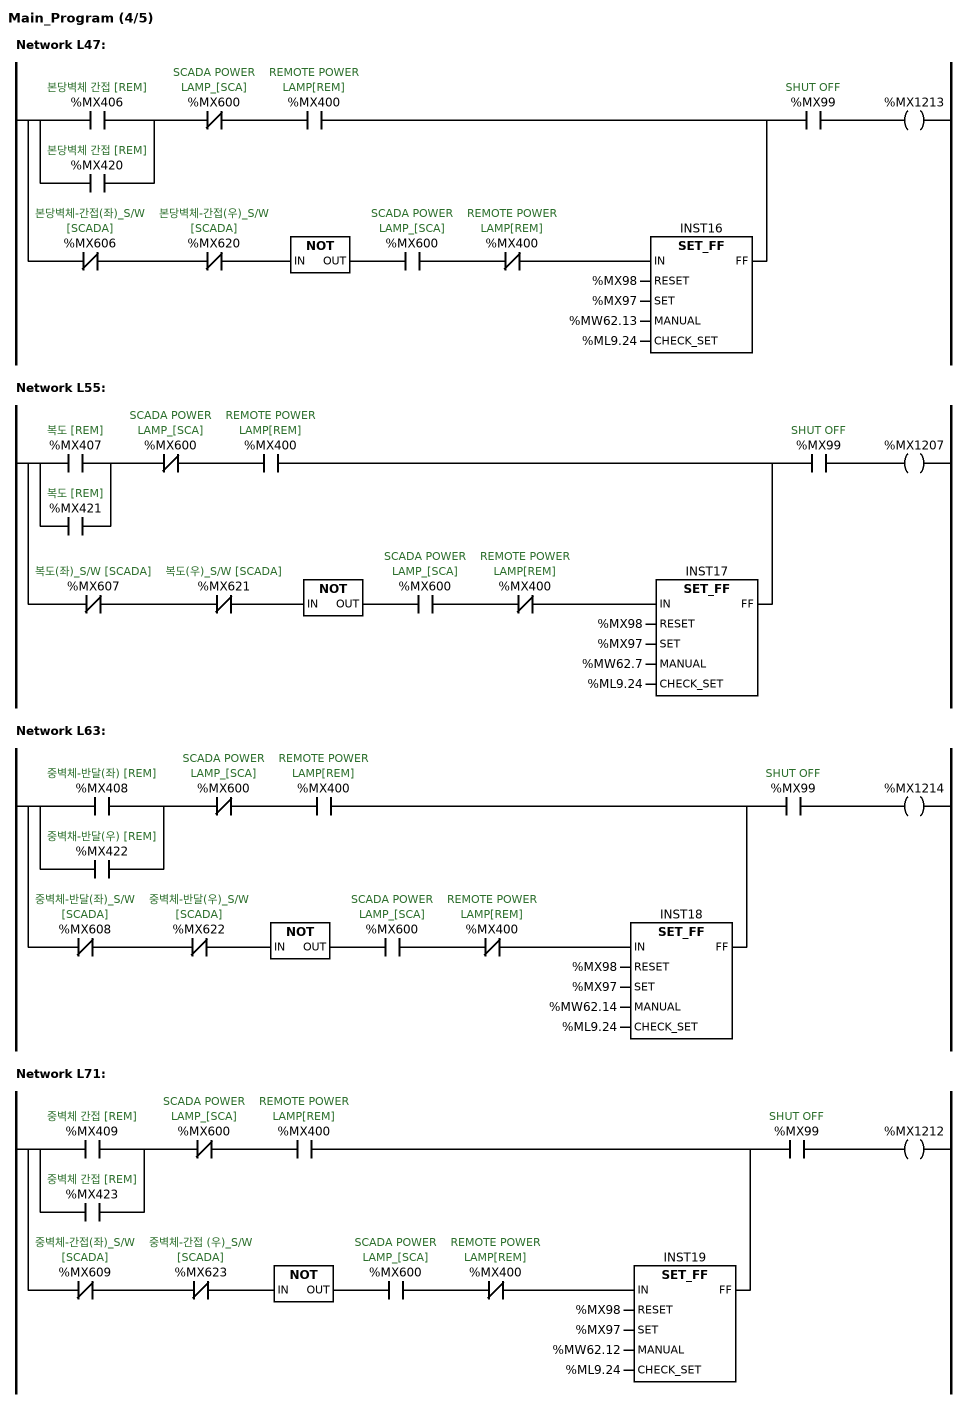
(* Rung L47 *)
INST16(IN := (NOT (NOT %MX606 AND NOT %MX620)) AND %MX600 AND NOT %MX400, RESET := %MX98, SET := %MX97, MANUAL := %MW62.13, CHECK_SET := %ML9.24);
%MX1213 := (((%MX406 OR %MX420) AND NOT %MX600 AND %MX400) OR INST16.FF) AND %MX99;
(* Rung L55 *)
INST17(IN := (NOT (NOT %MX607 AND NOT %MX621)) AND %MX600 AND NOT %MX400, RESET := %MX98, SET := %MX97, MANUAL := %MW62.7, CHECK_SET := %ML9.24);
%MX1207 := (((%MX407 OR %MX421) AND NOT %MX600 AND %MX400) OR INST17.FF) AND %MX99;
(* Rung L63 *)
INST18(IN := (NOT (NOT %MX608 AND NOT %MX622)) AND %MX600 AND NOT %MX400, RESET := %MX98, SET := %MX97, MANUAL := %MW62.14, CHECK_SET := %ML9.24);
%MX1214 := (((%MX408 OR %MX422) AND NOT %MX600 AND %MX400) OR INST18.FF) AND %MX99;
(* Rung L71 *)
INST19(IN := (NOT (NOT %MX609 AND NOT %MX623)) AND %MX600 AND NOT %MX400, RESET := %MX98, SET := %MX97, MANUAL := %MW62.12, CHECK_SET := %ML9.24);
%MX1212 := (((%MX409 OR %MX423) AND NOT %MX600 AND %MX400) OR INST19.FF) AND %MX99;

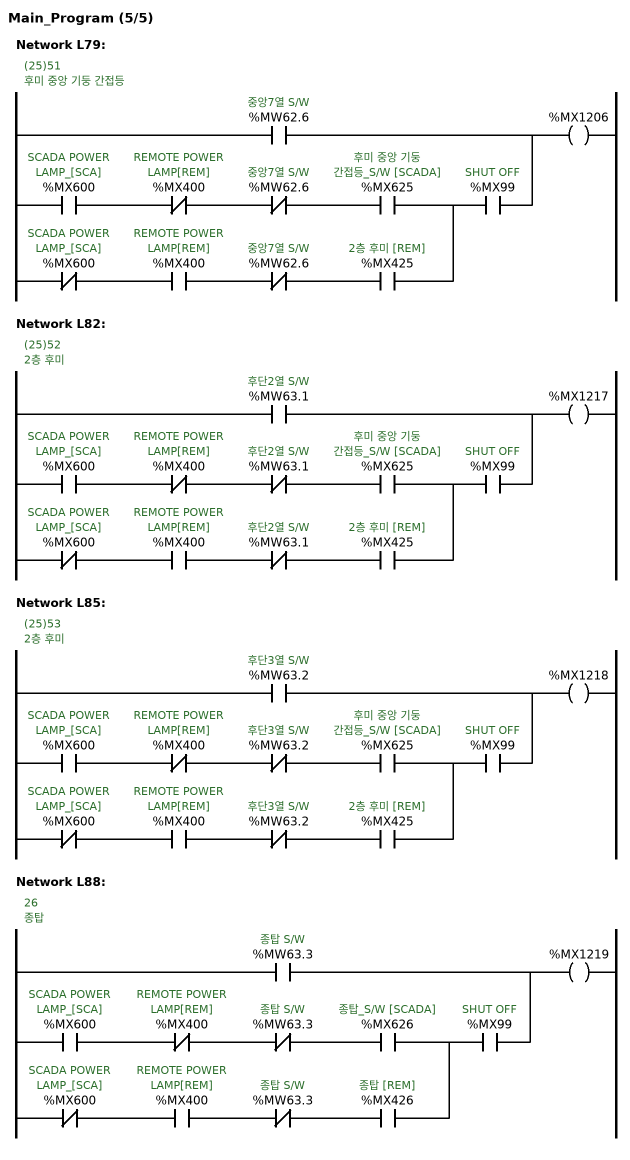
(* Rung L79 *)
%MX1206 := %MW62.6 OR (((%MX600 AND NOT %MX400 AND NOT %MW62.6 AND %MX625) OR (NOT %MX600 AND %MX400 AND NOT %MW62.6 AND %MX425)) AND %MX99);
(* (25)51 / 후미 중앙 기둥 간접등 *)
(* Rung L82 *)
%MX1217 := %MW63.1 OR (((%MX600 AND NOT %MX400 AND NOT %MW63.1 AND %MX625) OR (NOT %MX600 AND %MX400 AND NOT %MW63.1 AND %MX425)) AND %MX99);
(* (25)52 / 2층 후미 *)
(* Rung L85 *)
%MX1218 := %MW63.2 OR (((%MX600 AND NOT %MX400 AND NOT %MW63.2 AND %MX625) OR (NOT %MX600 AND %MX400 AND NOT %MW63.2 AND %MX425)) AND %MX99);
(* (25)53 / 2층 후미 *)
(* Rung L88 *)
%MX1219 := %MW63.3 OR (((%MX600 AND NOT %MX400 AND NOT %MW63.3 AND %MX626) OR (NOT %MX600 AND %MX400 AND NOT %MW63.3 AND %MX426)) AND %MX99);
(* 26 / 종탑 *)
END_PROGRAM

PROGRAM Input_Main (* task: 스캔 프로그램 *)

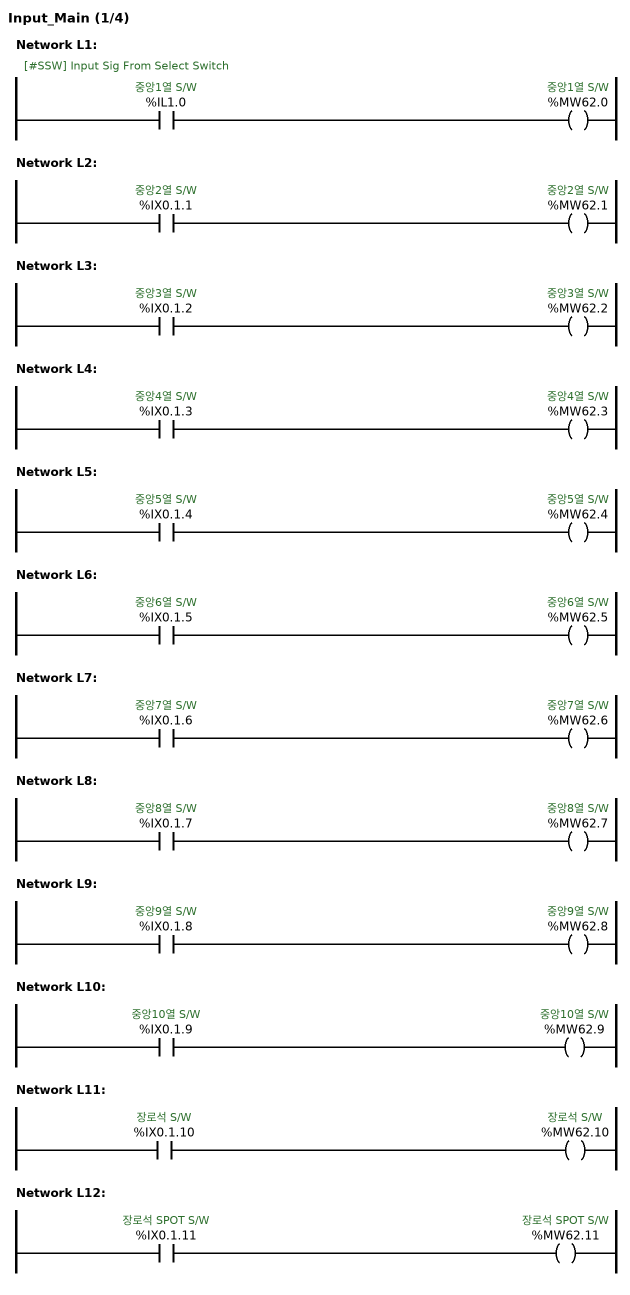
(* [#SSW] Input Sig From Select Switch *)
(* Rung L1 *)
%MW62.0 := %IL1.0;
(* Rung L2 *)
%MW62.1 := %IX0.1.1;
(* Rung L3 *)
%MW62.2 := %IX0.1.2;
(* Rung L4 *)
%MW62.3 := %IX0.1.3;
(* Rung L5 *)
%MW62.4 := %IX0.1.4;
(* Rung L6 *)
%MW62.5 := %IX0.1.5;
(* Rung L7 *)
%MW62.6 := %IX0.1.6;
(* Rung L8 *)
%MW62.7 := %IX0.1.7;
(* Rung L9 *)
%MW62.8 := %IX0.1.8;
(* Rung L10 *)
%MW62.9 := %IX0.1.9;
(* Rung L11 *)
%MW62.10 := %IX0.1.10;
(* Rung L12 *)
%MW62.11 := %IX0.1.11;

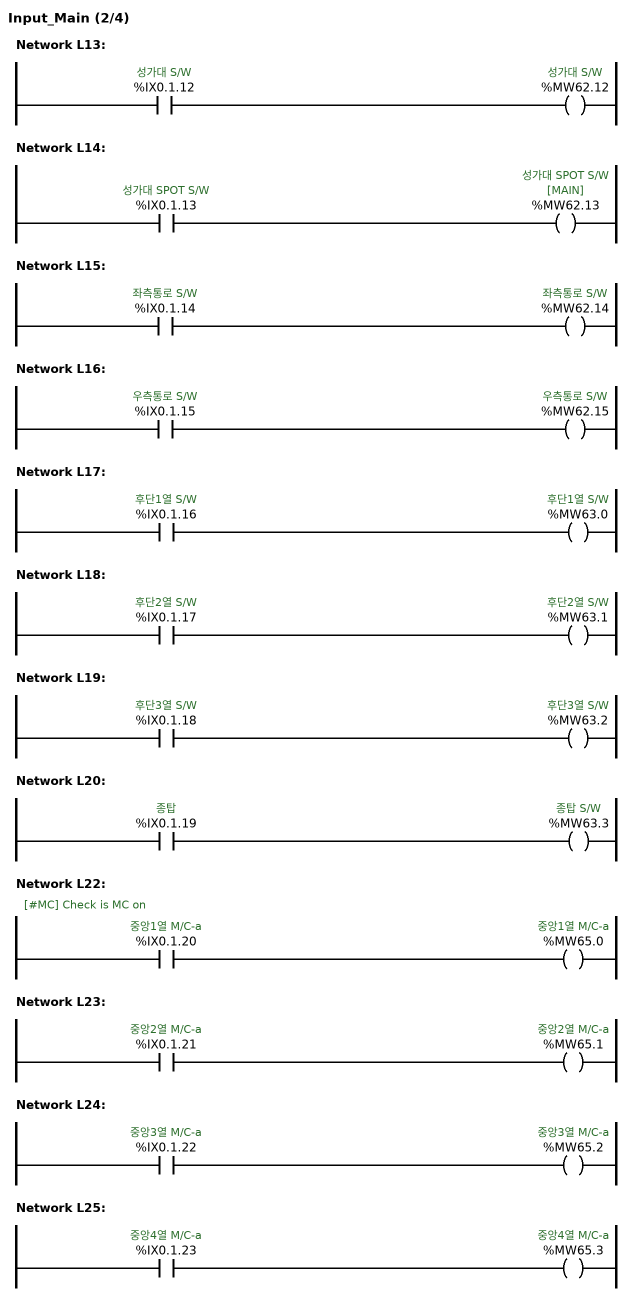
(* Rung L13 *)
%MW62.12 := %IX0.1.12;
(* Rung L14 *)
%MW62.13 := %IX0.1.13;
(* Rung L15 *)
%MW62.14 := %IX0.1.14;
(* Rung L16 *)
%MW62.15 := %IX0.1.15;
(* Rung L17 *)
%MW63.0 := %IX0.1.16;
(* Rung L18 *)
%MW63.1 := %IX0.1.17;
(* Rung L19 *)
%MW63.2 := %IX0.1.18;
(* Rung L20 *)
%MW63.3 := %IX0.1.19;
(* [#MC] Check is MC on *)
(* Rung L22 *)
%MW65.0 := %IX0.1.20;
(* Rung L23 *)
%MW65.1 := %IX0.1.21;
(* Rung L24 *)
%MW65.2 := %IX0.1.22;
(* Rung L25 *)
%MW65.3 := %IX0.1.23;

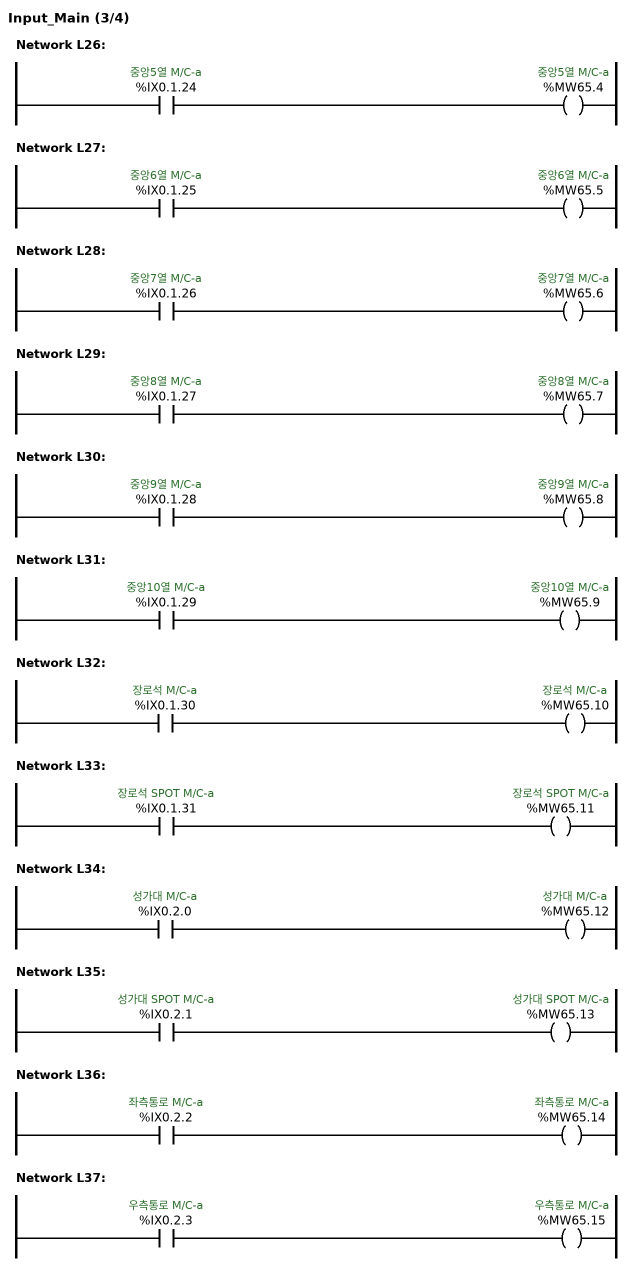
(* Rung L26 *)
%MW65.4 := %IX0.1.24;
(* Rung L27 *)
%MW65.5 := %IX0.1.25;
(* Rung L28 *)
%MW65.6 := %IX0.1.26;
(* Rung L29 *)
%MW65.7 := %IX0.1.27;
(* Rung L30 *)
%MW65.8 := %IX0.1.28;
(* Rung L31 *)
%MW65.9 := %IX0.1.29;
(* Rung L32 *)
%MW65.10 := %IX0.1.30;
(* Rung L33 *)
%MW65.11 := %IX0.1.31;
(* Rung L34 *)
%MW65.12 := %IX0.2.0;
(* Rung L35 *)
%MW65.13 := %IX0.2.1;
(* Rung L36 *)
%MW65.14 := %IX0.2.2;
(* Rung L37 *)
%MW65.15 := %IX0.2.3;

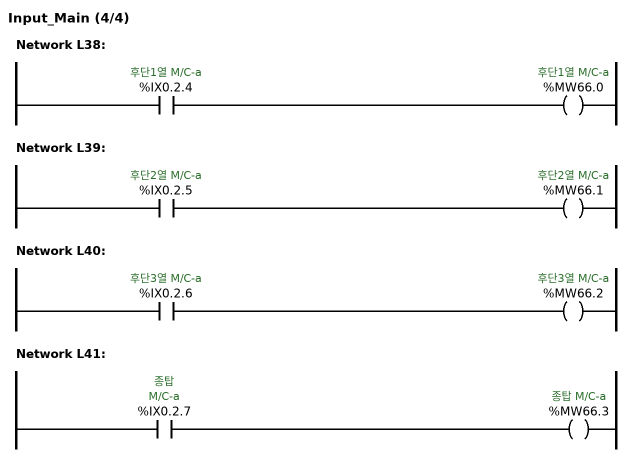
(* Rung L38 *)
%MW66.0 := %IX0.2.4;
(* Rung L39 *)
%MW66.1 := %IX0.2.5;
(* Rung L40 *)
%MW66.2 := %IX0.2.6;
(* Rung L41 *)
%MW66.3 := %IX0.2.7;
END_PROGRAM

PROGRAM Output-Main (* task: 스캔 프로그램 *)

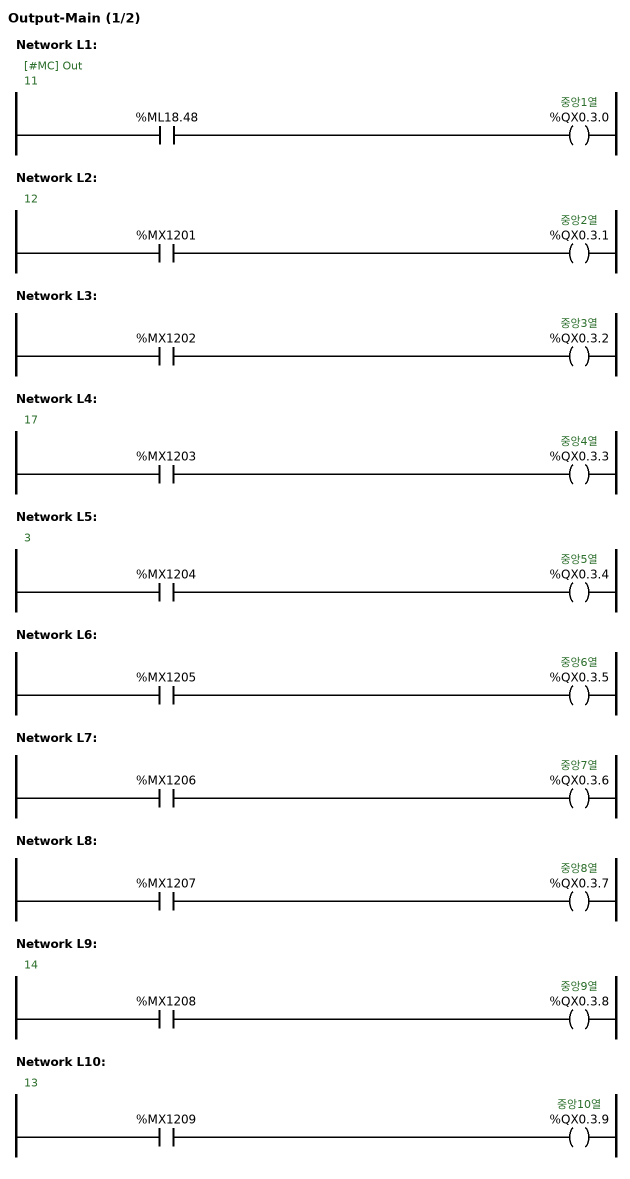
(* [#MC] Out *)
(* Rung L1 *)
%QX0.3.0 := %ML18.48;
(* 11 *)
(* Rung L2 *)
%QX0.3.1 := %MX1201;
(* 12 *)
(* Rung L3 *)
%QX0.3.2 := %MX1202;
(* Rung L4 *)
%QX0.3.3 := %MX1203;
(* 17 *)
(* Rung L5 *)
%QX0.3.4 := %MX1204;
(* 3 *)
(* Rung L6 *)
%QX0.3.5 := %MX1205;
(* Rung L7 *)
%QX0.3.6 := %MX1206;
(* Rung L8 *)
%QX0.3.7 := %MX1207;
(* Rung L9 *)
%QX0.3.8 := %MX1208;
(* 14 *)
(* Rung L10 *)
%QX0.3.9 := %MX1209;
(* 13 *)

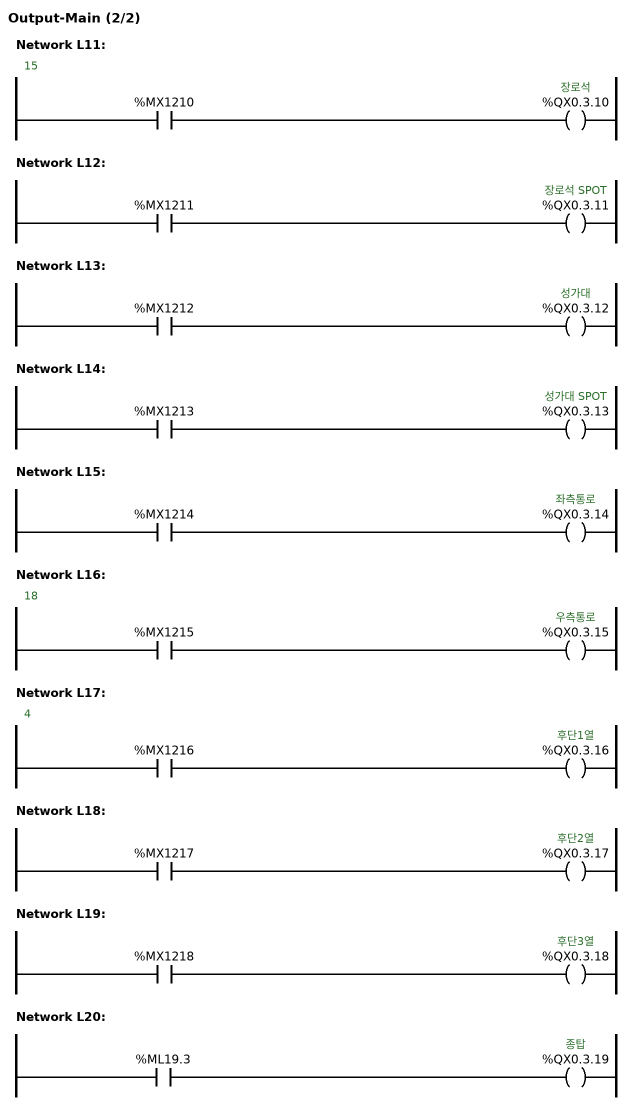
(* Rung L11 *)
%QX0.3.10 := %MX1210;
(* 15 *)
(* Rung L12 *)
%QX0.3.11 := %MX1211;
(* Rung L13 *)
%QX0.3.12 := %MX1212;
(* Rung L14 *)
%QX0.3.13 := %MX1213;
(* Rung L15 *)
%QX0.3.14 := %MX1214;
(* Rung L16 *)
%QX0.3.15 := %MX1215;
(* 18 *)
(* Rung L17 *)
%QX0.3.16 := %MX1216;
(* 4 *)
(* Rung L18 *)
%QX0.3.17 := %MX1217;
(* Rung L19 *)
%QX0.3.18 := %MX1218;
(* Rung L20 *)
%QX0.3.19 := %ML19.3;
END_PROGRAM

PROGRAM Alarm_Remote (* task: 스캔 프로그램 *)
VAR
    BUZZER : BOOL; (* BUZZER / SIG *)
    BZ_STOP : BOOL;
    FF : FF;
    INST : FF;
    INST1 : FF;
    INST2 : TON;
    INST9 : TMR_FLK;
END_VAR
VAR
    _p1 : BOOL;
    _t2 : BOOL;
END_VAR

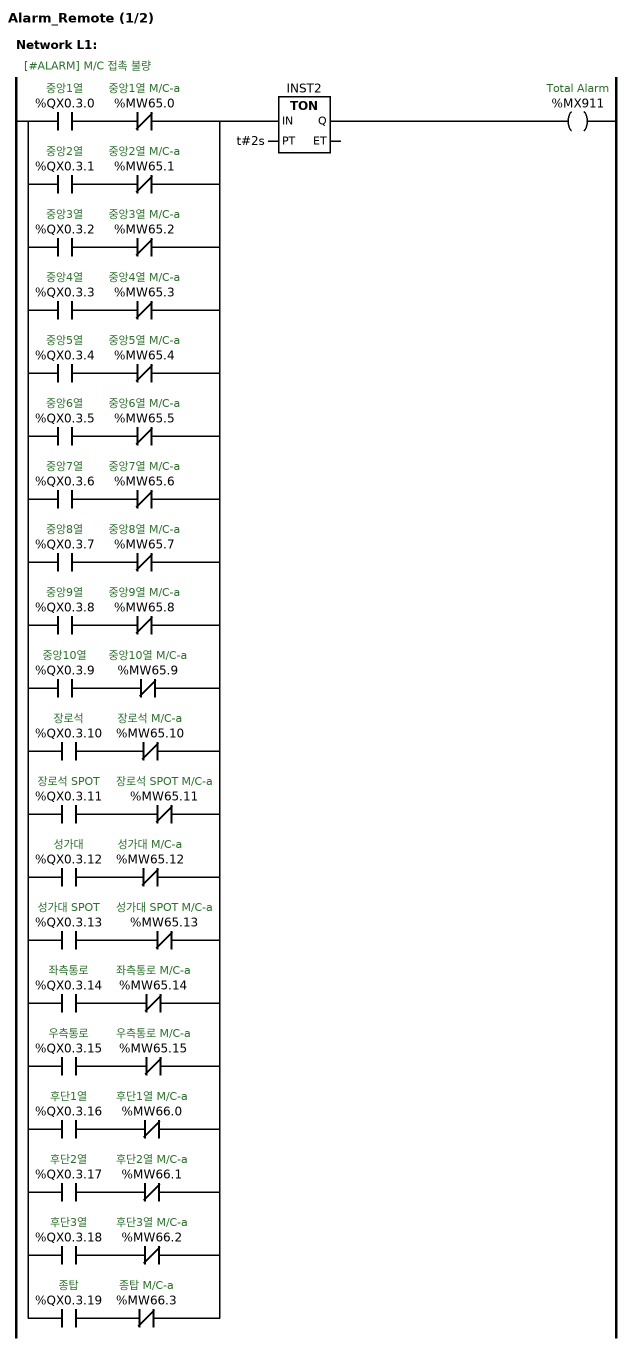
(* [#ALARM] M/C 접촉 불량 *)
(* Rung L1 *)
INST2(IN := (%QX0.3.0 AND NOT %MW65.0) OR (%QX0.3.1 AND NOT %MW65.1) OR (%QX0.3.2 AND NOT %MW65.2) OR (%QX0.3.3 AND NOT %MW65.3) OR (%QX0.3.4 AND NOT %MW65.4) OR (%QX0.3.5 AND NOT %MW65.5) OR (%QX0.3.6 AND NOT %MW65.6) OR (%QX0.3.7 AND NOT %MW65.7) OR (%QX0.3.8 AND NOT %MW65.8) OR (%QX0.3.9 AND NOT %MW65.9) OR (%QX0.3.10 AND NOT %MW65.10) OR (%QX0.3.11 AND NOT %MW65.11) OR (%QX0.3.12 AND NOT %MW65.12) OR (%QX0.3.13 AND NOT %MW65.13) OR (%QX0.3.14 AND NOT %MW65.14) OR (%QX0.3.15 AND NOT %MW65.15) OR (%QX0.3.16 AND NOT %MW66.0) OR (%QX0.3.17 AND NOT %MW66.1) OR (%QX0.3.18 AND NOT %MW66.2) OR (%QX0.3.19 AND NOT %MW66.3), PT := t#2s);
%MX911 := INST2.Q;

